{attribute 'GeneratedUsingTerminal: EK1122-0000-0018'}
{attribute addProperty BoxType "EK1122-0000-0018"}
{attribute addProperty Id "Beckhoff_EKx9xxsub_EK1100EK1100_1FC0878B2A_0001_EK1960_0000_0019EK1960_14394C51142A_0002_EK1960_0000_0021EK1960_9900B192138A_0003_EK1960_0008_0019EK1960_14394C51142A_0004_EK1960_0008_0021EK1960_9900B192138A_0005_EK1960_2600_0019EK1960_BAE25DEC148A_0006_EK1960_2600_0021EK1960_2415CDAE148A_0007_EK1960_2608_0019EK1960_BAE25DEC148A_0008_EK1960_2608_0021EK1960_2415CDAE148"}
{attribute addProperty CRC "1103075498"}
{attribute addProperty Size "1154"}
TYPE Beckhoff_EKx9xxEK1122_41BF98AA EXTENDS EK1122_1FC0878B :
STRUCT
	{attribute addProperty Name "Beckhoff EKx9xxsub EK1100"}
	{attribute addProperty PreviousPort "Beckhoff EKx9xxEK1122 : D"}
	Beckhoff_EKx9xxsub_EK1100 : EK1100_1FC0878B;
	{attribute addProperty Name "A_0001(EK1960-0000-0019)"}
	{attribute addProperty PreviousPort "Beckhoff EKx9xxsub EK1100 : C"}
	A_0001_EK1960_0000_0019 : EK1960_14394C51;
	{attribute addProperty Name "A_0002(EK1960-0000-0021)"}
	{attribute addProperty PreviousPort "A_0001(EK1960-0000-0019) : C"}
	A_0002_EK1960_0000_0021 : EK1960_9900B192;
	{attribute addProperty Name "A_0003(EK1960-0008-0019)"}
	{attribute addProperty PreviousPort "A_0002(EK1960-0000-0021) : C"}
	A_0003_EK1960_0008_0019 : EK1960_14394C51;
	{attribute addProperty Name "A_0004(EK1960-0008-0021)"}
	{attribute addProperty PreviousPort "A_0003(EK1960-0008-0019) : C"}
	A_0004_EK1960_0008_0021 : EK1960_9900B192;
	{attribute addProperty Name "A_0005(EK1960-2600-0019)"}
	{attribute addProperty PreviousPort "A_0004(EK1960-0008-0021) : C"}
	A_0005_EK1960_2600_0019 : EK1960_BAE25DEC;
	{attribute addProperty Name "A_0006(EK1960-2600-0021)"}
	{attribute addProperty PreviousPort "A_0005(EK1960-2600-0019) : C"}
	A_0006_EK1960_2600_0021 : EK1960_2415CDAE;
	{attribute addProperty Name "A_0007(EK1960-2608-0019)"}
	{attribute addProperty PreviousPort "A_0006(EK1960-2600-0021) : C"}
	A_0007_EK1960_2608_0019 : EK1960_BAE25DEC;
	{attribute addProperty Name "A_0008(EK1960-2608-0021)"}
	{attribute addProperty PreviousPort "A_0007(EK1960-2608-0019) : C"}
	A_0008_EK1960_2608_0021 : EK1960_2415CDAE;
END_STRUCT
END_TYPE

(* stored: Version 1.2.0.0, ProductVersion 3.1.4024.9
   DUT Beckhoff_EKx9xxEK1122_41BF98AA: Id {d8b155b2-2ae4-4d93-b336-ddb602b6c18f} *)
